TYPE ST_StationToTc3Hmi :
STRUCT
	stStationName			: ST_Text;	//example -> station 001
	
	//astButton				: ARRAY[0..CONST.iMaxIdxLocalButton] OF ST_HMI_BUTTON_OUT; //programmer defined buttons
	
	//stCounter				: ARRAY[0..CONST.iMaxIdxCounter] OF ST_Counter_Item_String;
	//stEingabeStatusColor	: ST_HMI_COLOR_STRING;
	//stEingabeStatus			: ST_Text;
	
END_STRUCT
END_TYPE

(* stored: Version 1.1.0.1, ProductVersion 3.1.4024.12
   DUT ST_StationToTc3Hmi: Id {810f8068-ed7b-4cd6-a54b-448bdb649440} *)
